TYPE ref_XYZ :
STRUCT
	x : LREAL ;
	y : LREAL ;
	z : LREAL ;
END_STRUCT
END_TYPE

(* stored: Version 1.1.0.1, ProductVersion 3.1.4024.11
   DUT ref_XYZ: Id {adc599e0-a1d9-496b-af09-4f02c477e488} *)
